(* IEC 61131-3 sources: POC_HINCAPIE/Project/SIEMENS/DIGSI/Guadalupe/TMP/CFC/7344242.18124 (part 2) *)

     AND10_9             (X1 := OR10_7.Y,
                          X2 := AND10_6.Y,
                          X3 := 1,
                          X4 := 1,
                          X5 := 1,
                          X6 := 1,
                          X7 := 1,
                          X8 := 1,
                          X9 := 1,
                          X10 := 1);

     AND10_10            (X1 := AND10_2.Y,
                          X2 := AND10_6.Y,
                          X3 := 1,
                          X4 := 1,
                          X5 := 1,
                          X6 := 1,
                          X7 := 1,
                          X8 := 1,
                          X9 := 1,
                          X10 := 1);

     AND10_11            (X1 := AND10_6.Y,
                          X2 := AND10_3.Y,
                          X3 := 1,
                          X4 := 1,
                          X5 := 1,
                          X6 := 1,
                          X7 := 1,
                          X8 := 1,
                          X9 := 1,
                          X10 := 1);

     OR10_12             (X1 := AND10_9.Y,
                          X2 := AND10_8.Y,
                          X3 := 0,
                          X4 := 0,
                          X5 := 0,
                          X6 := 0,
                          X7 := 0,
                          X8 := 0,
                          X9 := 0,
                          X10 := 0);

     AND10_13            (X1 := EXV_SPS_0144.VAL(* POSITION := 39*79: SIZE := 32* -1:   *) ,
                          X2 := EXV_SPS_0148.VAL(* POSITION := 40*80: SIZE := 31* -1:   *) ,
                          X3 := OR10_1.Y,
                          X4 := 1,
                          X5 := 1,
                          X6 := 1,
                          X7 := 1,
                          X8 := 1,
                          X9 := 1,
                          X10 := 1);

     EXV_SPS_0123        (LNK := 123,
                          VAL := AND10_3.Y(* POSITION := 53*59: SIZE := 32* -1:   *) );
     EXV_SPS_0124        (LNK := 124,
                          VAL := AND10_11.Y(* POSITION := 119*19: SIZE := 34* -1:   *) );
     EXV_SPS_0125        (LNK := 125,
                          VAL := AND10_2.Y(* POSITION := 65*7: SIZE := 32* -1:   *) );
     EXV_SPS_0126        (LNK := 126,
                          VAL := AND10_10.Y(* POSITION := 119*12: SIZE := 34* -1:   *) );
     EXV_SPS_0127        (LNK := 127,
                          VAL := OR10_7.Y(* POSITION := 117*26: SIZE := 31* -1:   *) );
     EXV_SPS_0128        (LNK := 128,
                          VAL := AND10_9.Y(* POSITION := 117*37: SIZE := 34* -1:   *) );
     EXV_SPS_0129        (LNK := 129,
                          VAL := OR10_12.Y(* POSITION := 112*56: SIZE := 34* -1:   *) );
     EXV_SPS_0130        (LNK := 130,
                          VAL := AND10_8.Y(* POSITION := 93*67: SIZE := 32* -1:   *) );
     EXV_SPS_0131        (LNK := 131,
                          VAL := AND10_13.Y(* POSITION := 96*79: SIZE := 29* -1:   *) );
     EXV_SPS_0142        (LNK := 142,
                          VAL := AND10_8.Y(* POSITION := 93*66: SIZE := 34* -1:   *) );
     EXV_SPS_0143        (LNK := 143,
                          VAL := AND10_9.Y(* POSITION := 117*36: SIZE := 35* -1:   *) );
     EXV_SPS_0147        (LNK := 147,
                          VAL := OR10_1.Y(* POSITION := 97*87: SIZE := 31* -1:   *) );
     EXV_SPS_0149        (LNK := 149,
                          VAL := OR10_12.Y(* POSITION := 110*55: SIZE := 38* -1:   *) );
     EXV_SPS_0151        (LNK := 151,
                          VAL := AND10_5.Y(* POSITION := -1*-1: SIZE := 33* -1:   *) );

(* COMMENT_TEXT;{X=70,Y=2};{Width=33, Height=2};FontSize := 12,LineColor := 0,LineWidth := 0,Alignment := Near,AutoWrap := True,BackColor := -16711681,Background := False,TextColor := 0,WallpaperGamma := 100,PartitionID := 1,;Enclavamiento Cierre Interruptor de 13.8 kV *)
(* COMMENT_TEXT;{X=12,Y=6};{Width=21, Height=2};FontSize := 12,LineColor := 0,LineWidth := 0,Alignment := Near,AutoWrap := True,BackColor := -16711681,Background := False,TextColor := 0,WallpaperGamma := 100,PartitionID := 1,;Interruptor Mantenimiento *)
(* COMMENT_TEXT;{X=18,Y=46};{Width=17, Height=2};FontSize := 12,LineColor := 0,LineWidth := 0,Alignment := Near,AutoWrap := True,BackColor := -16711681,Background := False,TextColor := 0,WallpaperGamma := 100,PartitionID := 1,;Interruptor Operación *)
(* COMMENT_TEXT;{X=33,Y=61};{Width=37, Height=2};FontSize := 12,LineColor := 0,LineWidth := 0,Alignment := Near,AutoWrap := True,BackColor := -16711681,Background := False,TextColor := 0,WallpaperGamma := 100,PartitionID := 1,;Enclavamientos Apertura Interruptor de 13.8 kV *)

END_PROGRAM

                                                  (* ---------- Program : CHART_dc33a26f_dd72_4905_a63e_bf494be4a4b3 ----------  *)

PROGRAM CHART_dc33a26f_dd72_4905_a63e_bf494be4a4b3
{COMMENT := "Enclavamiento Q1 - Q2";DESC := "";}
(* ChartLayout;PageSize := A4,Rows := 3,Columns := 2,MarginMode := WithoutMargins,MarginSize := 37,MarginLines := 1 *)
(* PartitionInfo;Id := 1,Name := Partition_1,Comment :=   *)
VAR

     (* IO_IOVISIBILITY;OR10_1;X3:X4:X5:X6:X7:X8:X9:X10: *)

     (* PartitionInfo;PartitionID OR10_1;1  *)
OR10_1          { COMMENT := 'or10_4'; POSITION := 49,39; SIZE := 12, 12; } :OR10;

     (* IO_IOVISIBILITY;OR10_2;X3:X4:X5:X6:X7:X8:X9:X10: *)

     (* PartitionInfo;PartitionID OR10_2;1  *)
OR10_2          { COMMENT := 'or10_9'; POSITION := 49,113; SIZE := 12, 12; } :OR10;

     (* IO_IOVISIBILITY;AND10_3;X3:X4:X5:X6:X7:X8:X9:X10: *)

     (* PartitionInfo;PartitionID AND10_3;1  *)
AND10_3         { COMMENT := 'and10_1'; POSITION := 48,6; SIZE := 12, 12; } :AND10;

     (* IO_IOVISIBILITY;AND10_4;X4:X5:X6:X7:X8:X9:X10: *)

     (* PartitionInfo;PartitionID AND10_4;1  *)
AND10_4         { COMMENT := 'and10_2'; POSITION := 48,14; SIZE := 12, 12; } :AND10;

     (* IO_IOVISIBILITY;AND10_5;X3:X4:X5:X6:X7:X8:X9:X10: *)

     (* PartitionInfo;PartitionID AND10_5;1  *)
AND10_5         { COMMENT := 'and10_5'; POSITION := 49,81; SIZE := 12, 12; } :AND10;

     (* IO_IOVISIBILITY;AND10_6;X4:X5:X6:X7:X8:X9:X10: *)

     (* PartitionInfo;PartitionID AND10_6;1  *)
AND10_6         { COMMENT := 'and10_6'; POSITION := 49,89; SIZE := 12, 12; } :AND10;

     (* IO_IOVISIBILITY;AND10_7;X6:X7:X8:X9:X10: *)

     (* PartitionInfo;PartitionID AND10_7;1  *)
AND10_7         { COMMENT := 'and10_4'; POSITION := 49,29; SIZE := 12, 12; } :AND10;

     (* IO_IOVISIBILITY;AND10_8;X6:X7:X8:X9:X10: *)

     (* PartitionInfo;PartitionID AND10_8;1  *)
AND10_8         { COMMENT := 'and10_22'; POSITION := 49,103; SIZE := 12, 12; } :AND10;

     (* IO_IOVISIBILITY;OR10_9;X3:X4:X5:X6:X7:X8:X9:X10: *)

     (* PartitionInfo;PartitionID OR10_9;1  *)
OR10_9          { COMMENT := 'or10_1'; POSITION := 70,22; SIZE := 12, 12; } :OR10;

     (* IO_IOVISIBILITY;OR10_10;X3:X4:X5:X6:X7:X8:X9:X10: *)

     (* PartitionInfo;PartitionID OR10_10;1  *)
OR10_10         { COMMENT := 'or10_2'; POSITION := 69,95; SIZE := 12, 12; } :OR10;

     (* IO_IOVISIBILITY;AND10_11;X3:X4:X5:X6:X7:X8:X9:X10: *)

     (* PartitionInfo;PartitionID AND10_11;1  *)
AND10_11        { COMMENT := 'and10_3'; POSITION := 89,28; SIZE := 12, 12; } :AND10;

     (* IO_IOVISIBILITY;AND10_12;X3:X4:X5:X6:X7:X8:X9:X10: *)

     (* PartitionInfo;PartitionID AND10_12;1  *)
AND10_12        { COMMENT := 'and10_7'; POSITION := 93,102; SIZE := 12, 12; } :AND10;

     (* 0152 - GDL69TRF2BCU_.Application.FG1_UserDef.FB2_Universal.PerQ1 *)
     EXV_SPS_0152   {COMMENT := "GDL69TRF2BCU_.Application.FG1_UserDef.FB2_Universal.PerQ1";DESC := "0##Application#Usuario#Logicas#Permisivo Q1##1";}:OEXV_BO_SPS;

     (* 0153 - GDL69TRF2BCU_.Application.FG1_Switch.FB1_XSWI.Pos.DPC_StatusOff *)
     EXV_SPS_0153   {COMMENT := "GDL69TRF2BCU_.Application.FG1_Switch.FB1_XSWI.Pos.DPC_StatusOff";DESC := "0##Application#6T4-Q1#Disconnector#Position#open##1";}:IEXV_SPS_BO;

     (* 0154 - GDL69TRF2BCU_.Application.FG1_Breaker_3pol.FB1_XCBR.Pos.DPC_StatusOff *)
     EXV_SPS_0154   {COMMENT := "GDL69TRF2BCU_.Application.FG1_Breaker_3pol.FB1_XCBR.Pos.DPC_StatusOff";DESC := "0##Application#6T4-Q0#Circuit break.#Position#open##1";}:IEXV_SPS_BO;

     (* 0155 - GDL69TRF2BCU_.Application.FG1_Switch.FB1_XSWI.Pos.DPC_StatusOn *)
     EXV_SPS_0155   {COMMENT := "GDL69TRF2BCU_.Application.FG1_Switch.FB1_XSWI.Pos.DPC_StatusOn";DESC := "0##Application#6T4-Q1#Disconnector#Position#closed##1";}:IEXV_SPS_BO;

     (* 0156 - GDL69TRF2BCU_.Application.FG2_Switch.FB1_XSWI.Pos.DPC_StatusOn *)
     EXV_SPS_0156   {COMMENT := "GDL69TRF2BCU_.Application.FG2_Switch.FB1_XSWI.Pos.DPC_StatusOn";DESC := "0##Application#6T4-Q2#Disconnector#Position#closed##1";}:IEXV_SPS_BO;

     (* 0157 - GDL69TRF2BCU_.Application.FG2_Switch.FB1_XSWI.Pos.DPC_StatusOff *)
     EXV_SPS_0157   {COMMENT := "GDL69TRF2BCU_.Application.FG2_Switch.FB1_XSWI.Pos.DPC_StatusOff";DESC := "0##Application#6T4-Q2#Disconnector#Position#open##1";}:IEXV_SPS_BO;

     (* 0158 - GDL69TRF2BCU_.Application.FG1_Switch.FB1_CILO.EnaOpnFix *)
     EXV_SPS_0158   {COMMENT := "GDL69TRF2BCU_.Application.FG1_Switch.FB1_CILO.EnaOpnFix";DESC := "0##Application#6T4-Q1#Interlocking#>Enable opening(fixed)##1";}:OEXV_BO_SPS;

     (* 0159 - GDL69TRF2BCU_.Application.FG1_Switch.FB1_CILO.EnaClsFix *)
     EXV_SPS_0159   {COMMENT := "GDL69TRF2BCU_.Application.FG1_Switch.FB1_CILO.EnaClsFix";DESC := "0##Application#6T4-Q1#Interlocking#>Enable closing (fixed)##1";}:OEXV_BO_SPS;

     (* 0160 - GDL69TRF2BCU_.Application.FG1_UserDef.FB1_Universal.SPS43 *)
     EXV_SPS_0160   {COMMENT := "GDL69TRF2BCU_.Application.FG1_UserDef.FB1_Universal.SPS43";DESC := "0##Application#Usuario#Entradas#Selector Remoto Q1##1";}:IEXV_SPS_BO;

     (* 0161 - GDL69TRF2BCU_.Application.FG1_UserDef.FB1_Universal.FaVcdQ1 *)
     EXV_SPS_0161   {COMMENT := "GDL69TRF2BCU_.Application.FG1_UserDef.FB1_Universal.FaVcdQ1";DESC := "0##Application#Usuario#Entradas#FVCD Q1##1";}:IEXV_SPS_BO;

     (* 0162 - GDL69TRF2BCU_.Application.FG1_UserDef.FB1_Universal.FaVcdSecc *)
     EXV_SPS_0162   {COMMENT := "GDL69TRF2BCU_.Application.FG1_UserDef.FB1_Universal.FaVcdSecc";DESC := "0##Application#Usuario#Entradas#FVCD Cto Control Seccionadores##1";}:IEXV_SPS_BO;

     (* 0163 - GDL69TRF2BCU_.Application.FG2_Switch.FB1_CILO.EnaOpnFix *)
     EXV_SPS_0163   {COMMENT := "GDL69TRF2BCU_.Application.FG2_Switch.FB1_CILO.EnaOpnFix";DESC := "0##Application#6T4-Q2#Interlocking#>Enable opening(fixed)##1";}:OEXV_BO_SPS;

     (* 0164 - GDL69TRF2BCU_.Application.FG2_Switch.FB1_CILO.EnaClsFix *)
     EXV_SPS_0164   {COMMENT := "GDL69TRF2BCU_.Application.FG2_Switch.FB1_CILO.EnaClsFix";DESC := "0##Application#6T4-Q2#Interlocking#>Enable closing (fixed)##1";}:OEXV_BO_SPS;

     (* 0165 - GDL69TRF2BCU_.Application.FG1_UserDef.FB1_Universal.FaVcdQ2 *)
     EXV_SPS_0165   {COMMENT := "GDL69TRF2BCU_.Application.FG1_UserDef.FB1_Universal.FaVcdQ2";DESC := "0##Application#Usuario#Entradas#FVCD Q2##1";}:IEXV_SPS_BO;

     (* 0166 - GDL69TRF2BCU_.Application.FG1_UserDef.FB1_Universal.SPS49 *)
     EXV_SPS_0166   {COMMENT := "GDL69TRF2BCU_.Application.FG1_UserDef.FB1_Universal.SPS49";DESC := "0##Application#Usuario#Entradas#Selector Remoto Q2##1";}:IEXV_SPS_BO;

     (* 0167 - GDL69TRF2BCU_.Application.FG1_Breaker_3pol.FB1_XCBR.Pos.DPC_StatusOn *)
     EXV_SPS_0167   {COMMENT := "GDL69TRF2BCU_.Application.FG1_Breaker_3pol.FB1_XCBR.Pos.DPC_StatusOn";DESC := "0##Application#6T4-Q0#Circuit break.#Position#closed##1";}:IEXV_SPS_BO;

     (* 0168 - GDL69TRF2BCU_.Application.FG1_UserDef.FB1_Universal.SPS113 *)
     EXV_SPS_0168   {COMMENT := "GDL69TRF2BCU_.Application.FG1_UserDef.FB1_Universal.SPS113";DESC := "0##Application#Usuario#Entradas#Bahia Acople Cerrada##1";}:IEXV_SPS_BO;

     (* 0169 - GDL69TRF2BCU_.Application.FG1_UserDef.FB2_Universal.PerQ1AcpCrdo *)
     EXV_SPS_0169   {COMMENT := "GDL69TRF2BCU_.Application.FG1_UserDef.FB2_Universal.PerQ1AcpCrdo";DESC := "0##Application#Usuario#Logicas#Permisivo Q1 Acople Cerrado##1";}:OEXV_BO_SPS;

     (* 0170 - GDL69TRF2BCU_.Application.FG1_UserDef.FB2_Universal.OrQ1 *)
     EXV_SPS_0170   {COMMENT := "GDL69TRF2BCU_.Application.FG1_UserDef.FB2_Universal.OrQ1";DESC := "0##Application#Usuario#Logicas#Or Q1##1";}:OEXV_BO_SPS;

     (* 0171 - GDL69TRF2BCU_.Application.FG1_UserDef.FB2_Universal.PerQ1Gral *)
     EXV_SPS_0171   {COMMENT := "GDL69TRF2BCU_.Application.FG1_UserDef.FB2_Universal.PerQ1Gral";DESC := "0##Application#Usuario#Logicas#Permisivo General Q1##1";}:OEXV_BO_SPS;

     (* 0172 - GDL69TRF2BCU_.Application.FG1_UserDef.FB2_Universal.OrQ2 *)
     EXV_SPS_0172   {COMMENT := "GDL69TRF2BCU_.Application.FG1_UserDef.FB2_Universal.OrQ2";DESC := "0##Application#Usuario#Logicas#Or Q2##1";}:OEXV_BO_SPS;

     (* 0173 - GDL69TRF2BCU_.Application.FG1_UserDef.FB2_Universal.PerQ2AcpCrdo *)
     EXV_SPS_0173   {COMMENT := "GDL69TRF2BCU_.Application.FG1_UserDef.FB2_Universal.PerQ2AcpCrdo";DESC := "0##Application#Usuario#Logicas#Permisivo Q2 Acople Cerrado##1";}:OEXV_BO_SPS;

     (* 0174 - GDL69TRF2BCU_.Application.FG1_UserDef.FB2_Universal.PerQ2Gral *)
     EXV_SPS_0174   {COMMENT := "GDL69TRF2BCU_.Application.FG1_UserDef.FB2_Universal.PerQ2Gral";DESC := "0##Application#Usuario#Logicas#Permisivo General Q2##1";}:OEXV_BO_SPS;

     (* 0175 - GDL69TRF2BCU_.Application.FG1_UserDef.FB2_Universal.PerQ2 *)
     EXV_SPS_0175   {COMMENT := "GDL69TRF2BCU_.Application.FG1_UserDef.FB2_Universal.PerQ2";DESC := "0##Application#Usuario#Logicas#Permisivo Q2##1";}:OEXV_BO_SPS;

     (* 0176 - GDL69TRF2BCU_.Application.FG1_UserDef.FB1_Universal.ManiInsertQ1 *)
     EXV_SPS_0176   {COMMENT := "GDL69TRF2BCU_.Application.FG1_UserDef.FB1_Universal.ManiInsertQ1";DESC := "0##Application#Usuario#Entradas#Manivela Insertada Q1##1";}:IEXV_SPS_BO;

     (* 0177 - GDL69TRF2BCU_.Application.FG1_UserDef.FB1_Universal.ManiInsertQ2 *)
     EXV_SPS_0177   {COMMENT := "GDL69TRF2BCU_.Application.FG1_UserDef.FB1_Universal.ManiInsertQ2";DESC := "0##Application#Usuario#Entradas#Manivela Insertada Q2##1";}:IEXV_SPS_BO;
END_VAR

     EXV_SPS_0153        (LNK := 153);

     EXV_SPS_0154        (LNK := 154);

     EXV_SPS_0155        (LNK := 155);

     EXV_SPS_0156        (LNK := 156);

     EXV_SPS_0157        (LNK := 157);

     EXV_SPS_0160        (LNK := 160);

     EXV_SPS_0161        (LNK := 161);

     EXV_SPS_0162        (LNK := 162);

     EXV_SPS_0165        (LNK := 165);

     EXV_SPS_0166        (LNK := 166);

     EXV_SPS_0167        (LNK := 167);

     EXV_SPS_0168        (LNK := 168);

     EXV_SPS_0176        (LNK := 176);

     EXV_SPS_0177        (LNK := 177);

     OR10_1              (X1 := EXV_SPS_0153.VAL(* POSITION := 13*42: SIZE := 30* -1:   *) ,
                          X2 := EXV_SPS_0155.VAL(* POSITION := 12*43: SIZE := 31* -1:   *) ,
                          X3 := 0,
                          X4 := 0,
                          X5 := 0,
                          X6 := 0,
                          X7 := 0,
                          X8 := 0,
                          X9 := 0,
                          X10 := 0);

     OR10_2              (X1 := EXV_SPS_0157.VAL(* POSITION := 13*116: SIZE := 30* -1:   *) ,
                          X2 := EXV_SPS_0156.VAL(* POSITION := 12*117: SIZE := 31* -1:   *) ,
                          X3 := 0,
                          X4 := 0,
                          X5 := 0,
                          X6 := 0,
                          X7 := 0,
                          X8 := 0,
                          X9 := 0,
                          X10 := 0);

     AND10_3             (X1 := EXV_SPS_0157.VAL(* POSITION := 12*9: SIZE := 30* -1:   *) ,
                          X2 := EXV_SPS_0154.VAL(* POSITION := 11*10: SIZE := 31* -1:   *) ,
                          X3 := 1,
                          X4 := 1,
                          X5 := 1,
                          X6 := 1,
                          X7 := 1,
                          X8 := 1,
                          X9 := 1,
                          X10 := 1);

     AND10_4             (X1 := EXV_SPS_0156.VAL(* POSITION := 11*17: SIZE := 31* -1:   *) ,
                          X2 := EXV_SPS_0167.VAL(* POSITION := 10*18: SIZE := 32* -1:   *) ,
                          X3 := EXV_SPS_0168.VAL(* POSITION := 10*19: SIZE := 32* -1:   *) ,
                          X4 := 1,
                          X5 := 1,
                          X6 := 1,
                          X7 := 1,
                          X8 := 1,
                          X9 := 1,
                          X10 := 1);

     AND10_5             (X1 := EXV_SPS_0153.VAL(* POSITION := 13*84: SIZE := 30* -1:   *) ,
                          X2 := EXV_SPS_0154.VAL(* POSITION := 12*85: SIZE := 31* -1:   *) ,
                          X3 := 1,
                          X4 := 1,
                          X5 := 1,
                          X6 := 1,
                          X7 := 1,
                          X8 := 1,
                          X9 := 1,
                          X10 := 1);

     AND10_6             (X1 := EXV_SPS_0155.VAL(* POSITION := 10*92: SIZE := 31* -1:   *) ,
                          X2 := EXV_SPS_0167.VAL(* POSITION := 9*93: SIZE := 32* -1:   *) ,
                          X3 := EXV_SPS_0168.VAL(* POSITION := 9*94: SIZE := 32* -1:   *) ,
                          X4 := 1,
                          X5 := 1,
                          X6 := 1,
                          X7 := 1,
                          X8 := 1,
                          X9 := 1,
                          X10 := 1);

     AND10_7             (X1 := EXV_SPS_0160.VAL(* POSITION := 10*32: SIZE := 31* -1:   *) ,
                          X2 := NOT EXV_SPS_0161.VAL(* POSITION := 16*33: SIZE := 25* -1:   *) ,
                          X3 := NOT EXV_SPS_0162.VAL(* POSITION := 4*34: SIZE := 37* -1:   *) ,
                          X4 := NOT EXV_SPS_0176.VAL(* POSITION := 9*35: SIZE := 32* -1:   *) ,
                          X5 := OR10_1.Y,
                          X6 := 1,
                          X7 := 1,
                          X8 := 1,
                          X9 := 1,
                          X10 := 1);

     AND10_8             (X1 := EXV_SPS_0166.VAL(* POSITION := -1*-1: SIZE := 31* -1:   *) ,
                          X2 := NOT EXV_SPS_0165.VAL(* POSITION := -1*-1: SIZE := 25* -1:   *) ,
                          X3 := NOT EXV_SPS_0162.VAL(* POSITION := -1*-1: SIZE := 37* -1:   *) ,
                          X4 := NOT EXV_SPS_0177.VAL(* POSITION := -1*-1: SIZE := 32* -1:   *) ,
                          X5 := OR10_2.Y,
                          X6 := 1,
                          X7 := 1,
                          X8 := 1,
                          X9 := 1,
                          X10 := 1);

     OR10_9              (X1 := AND10_3.Y,
                          X2 := AND10_4.Y,
                          X3 := 0,
                          X4 := 0,
                          X5 := 0,
                          X6 := 0,
                          X7 := 0,
                          X8 := 0,
                          X9 := 0,
                          X10 := 0);

     OR10_10             (X1 := AND10_5.Y,
                          X2 := AND10_6.Y,
                          X3 := 0,
                          X4 := 0,
                          X5 := 0,
                          X6 := 0,
                          X7 := 0,
                          X8 := 0,
                          X9 := 0,
                          X10 := 0);

     AND10_11            (X1 := OR10_9.Y,
                          X2 := AND10_7.Y,
                          X3 := 1,
                          X4 := 1,
                          X5 := 1,
                          X6 := 1,
                          X7 := 1,
                          X8 := 1,
                          X9 := 1,
                          X10 := 1);

     AND10_12            (X1 := OR10_10.Y,
                          X2 := AND10_8.Y,
                          X3 := 1,
                          X4 := 1,
                          X5 := 1,
                          X6 := 1,
                          X7 := 1,
                          X8 := 1,
                          X9 := 1,
                          X10 := 1);

     EXV_SPS_0152        (LNK := 152,
                          VAL := AND10_3.Y(* POSITION := 67*9: SIZE := 27* -1:   *) );
     EXV_SPS_0158        (LNK := 158,
                          VAL := AND10_11.Y(* POSITION := 108*33: SIZE := 34* -1:   *) );
     EXV_SPS_0159        (LNK := 159,
                          VAL := AND10_11.Y(* POSITION := 108*32: SIZE := 35* -1:   *) );
     EXV_SPS_0163        (LNK := 163,
                          VAL := AND10_12.Y(* POSITION := 112*106: SIZE := 34* -1:   *) );
     EXV_SPS_0164        (LNK := 164,
                          VAL := AND10_12.Y(* POSITION := 112*105: SIZE := 35* -1:   *) );
     EXV_SPS_0169        (LNK := 169,
                          VAL := AND10_4.Y(* POSITION := 68*17: SIZE := 35* -1:   *) );
     EXV_SPS_0170        (LNK := 170,
                          VAL := OR10_9.Y(* POSITION := 89*25: SIZE := 24* -1:   *) );
     EXV_SPS_0171        (LNK := 171,
                          VAL := AND10_11.Y(* POSITION := 108*31: SIZE := 31* -1:   *) );
     EXV_SPS_0172        (LNK := 172,
                          VAL := OR10_10.Y(* POSITION := 88*98: SIZE := 24* -1:   *) );
     EXV_SPS_0173        (LNK := 173,
                          VAL := AND10_6.Y(* POSITION := 68*92: SIZE := 35* -1:   *) );
     EXV_SPS_0174        (LNK := 174,
                          VAL := AND10_12.Y(* POSITION := 112*107: SIZE := 31* -1:   *) );
     EXV_SPS_0175        (LNK := 175,
                          VAL := AND10_5.Y(* POSITION := 68*84: SIZE := 27* -1:   *) );

(* COMMENT_TEXT;{X=43,Y=1};{Width=23, Height=2};FontSize := 12,LineColor := 0,LineWidth := 0,Alignment := Near,AutoWrap := True,BackColor := -16711681,Background := False,TextColor := 0,WallpaperGamma := 100,PartitionID := 1,;Enclavamiento Seccionador Q1 *)
(* COMMENT_TEXT;{X=45,Y=73};{Width=23, Height=2};FontSize := 12,LineColor := 0,LineWidth := 0,Alignment := Near,AutoWrap := True,BackColor := -16711681,Background := False,TextColor := 0,WallpaperGamma := 100,PartitionID := 1,;Enclavamiento Seccionador Q2 *)

END_PROGRAM

                                                  (* ---------- Program : CHART_Enclavamiento_Q9 ----------  *)

PROGRAM CHART_Enclavamiento_Q9
{COMMENT := "Enclavamiento Q9";DESC := "";}
(* ChartLayout;PageSize := A4,Rows := 3,Columns := 2,MarginMode := WithoutMargins,MarginSize := 37,MarginLines := 1 *)
(* PartitionInfo;Id := 1,Name := Partition_1,Comment :=   *)
VAR

     (* IO_IOVISIBILITY;OR10_1;X3:X4:X5:X6:X7:X8:X9:X10: *)

     (* PartitionInfo;PartitionID OR10_1;1  *)
OR10_1          { COMMENT := 'or10_5'; POSITION := 69,22; SIZE := 12, 12; } :OR10;

     (* IO_IOVISIBILITY;AND10_2;X7:X8:X9:X10: *)

     (* PartitionInfo;PartitionID AND10_2;1  *)
AND10_2         { COMMENT := 'and10_8'; POSITION := 69,11; SIZE := 12, 12; } :AND10;

     (* 0178 - GDL69TRF2BCU_.Application.FG1_UserDef.FB2_Universal.PerQ9 *)
     EXV_SPS_0178   {COMMENT := "GDL69TRF2BCU_.Application.FG1_UserDef.FB2_Universal.PerQ9";DESC := "0##Application#Usuario#Logicas#Permisivo Q9##1";}:OEXV_BO_SPS;

     (* 0179 - GDL69TRF2BCU_.Application.FG3_Switch.FB1_XSWI.Pos.DPC_StatusOff *)
     EXV_SPS_0179   {COMMENT := "GDL69TRF2BCU_.Application.FG3_Switch.FB1_XSWI.Pos.DPC_StatusOff";DESC := "0##Application#6T4-Q9#Disconnector#Position#open##1";}:IEXV_SPS_BO;

     (* 0180 - GDL69TRF2BCU_.Application.FG1_Breaker_3pol.FB1_XCBR.Pos.DPC_StatusOff *)
     EXV_SPS_0180   {COMMENT := "GDL69TRF2BCU_.Application.FG1_Breaker_3pol.FB1_XCBR.Pos.DPC_StatusOff";DESC := "0##Application#6T4-Q0#Circuit break.#Position#open##1";}:IEXV_SPS_BO;

     (* 0181 - GDL69TRF2BCU_.Application.FG3_Switch.FB1_XSWI.Pos.DPC_StatusOn *)
     EXV_SPS_0181   {COMMENT := "GDL69TRF2BCU_.Application.FG3_Switch.FB1_XSWI.Pos.DPC_StatusOn";DESC := "0##Application#6T4-Q9#Disconnector#Position#closed##1";}:IEXV_SPS_BO;

     (* 0182 - GDL69TRF2BCU_.Application.FG1_UserDef.FB1_Universal.FaVcdSecc *)
     EXV_SPS_0182   {COMMENT := "GDL69TRF2BCU_.Application.FG1_UserDef.FB1_Universal.FaVcdSecc";DESC := "0##Application#Usuario#Entradas#FVCD Cto Control Seccionadores##1";}:IEXV_SPS_BO;

     (* 0183 - GDL69TRF2BCU_.Application.FG1_UserDef.FB1_Universal.SPS55 *)
     EXV_SPS_0183   {COMMENT := "GDL69TRF2BCU_.Application.FG1_UserDef.FB1_Universal.SPS55";DESC := "0##Application#Usuario#Entradas#Selector Remoto Q9##1";}:IEXV_SPS_BO;

     (* 0184 - GDL69TRF2BCU_.Application.FG1_UserDef.FB1_Universal.FaVcdQ9 *)
     EXV_SPS_0184   {COMMENT := "GDL69TRF2BCU_.Application.FG1_UserDef.FB1_Universal.FaVcdQ9";DESC := "0##Application#Usuario#Entradas#FVCD Q9##1";}:IEXV_SPS_BO;

     (* 0185 - GDL69TRF2BCU_.Application.FG3_Switch.FB1_CILO.EnaClsFix *)
     EXV_SPS_0185   {COMMENT := "GDL69TRF2BCU_.Application.FG3_Switch.FB1_CILO.EnaClsFix";DESC := "0##Application#6T4-Q9#Interlocking#>Enable closing (fixed)##1";}:OEXV_BO_SPS;

     (* 0186 - GDL69TRF2BCU_.Application.FG3_Switch.FB1_CILO.EnaOpnFix *)
     EXV_SPS_0186   {COMMENT := "GDL69TRF2BCU_.Application.FG3_Switch.FB1_CILO.EnaOpnFix";DESC := "0##Application#6T4-Q9#Interlocking#>Enable opening(fixed)##1";}:OEXV_BO_SPS;

     (* 0187 - GDL69TRF2BCU_.Application.FG1_UserDef.FB1_Universal.ManiInsertQ9 *)
     EXV_SPS_0187   {COMMENT := "GDL69TRF2BCU_.Application.FG1_UserDef.FB1_Universal.ManiInsertQ9";DESC := "0##Application#Usuario#Entradas#Manivela Insertada Q9##1";}:IEXV_SPS_BO;
END_VAR

     EXV_SPS_0179        (LNK := 179);

     EXV_SPS_0180        (LNK := 180);

     EXV_SPS_0181        (LNK := 181);

     EXV_SPS_0182        (LNK := 182);

     EXV_SPS_0183        (LNK := 183);

     EXV_SPS_0184        (LNK := 184);

     EXV_SPS_0187        (LNK := 187);

     OR10_1              (X1 := EXV_SPS_0179.VAL(* POSITION := 33*25: SIZE := 30* -1:   *) ,
                          X2 := EXV_SPS_0181.VAL(* POSITION := 32*26: SIZE := 31* -1:   *) ,
                          X3 := 0,
                          X4 := 0,
                          X5 := 0,
                          X6 := 0,
                          X7 := 0,
                          X8 := 0,
                          X9 := 0,
                          X10 := 0);

     AND10_2             (X1 := EXV_SPS_0180.VAL(* POSITION := 32*14: SIZE := 31* -1:   *) ,
                          X2 := EXV_SPS_0183.VAL(* POSITION := 32*15: SIZE := 31* -1:   *) ,
                          X3 := NOT EXV_SPS_0184.VAL(* POSITION := 38*16: SIZE := 25* -1:   *) ,
                          X4 := NOT EXV_SPS_0182.VAL(* POSITION := 26*17: SIZE := 37* -1:   *) ,
                          X5 := NOT EXV_SPS_0187.VAL(* POSITION := -1*-1: SIZE := 32* -1:   *) ,
                          X6 := OR10_1.Y,
                          X7 := 1,
                          X8 := 1,
                          X9 := 1,
                          X10 := 1);

     EXV_SPS_0178        (LNK := 178,
                          VAL := AND10_2.Y(* POSITION := 88*16: SIZE := 27* -1:   *) );
     EXV_SPS_0185        (LNK := 185,
                          VAL := AND10_2.Y(* POSITION := 88*15: SIZE := 35* -1:   *) );
     EXV_SPS_0186        (LNK := 186,
                          VAL := AND10_2.Y(* POSITION := 88*14: SIZE := 34* -1:   *) );

(* COMMENT_TEXT;{X=63,Y=8};{Width=23, Height=2};FontSize := 12,LineColor := 0,LineWidth := 0,Alignment := Near,AutoWrap := True,BackColor := -16711681,Background := False,TextColor := 0,WallpaperGamma := 100,PartitionID := 1,;Enclavamiento Seccionador Q9 *)

END_PROGRAM

CONFIGURATION  PLC_CONTROL
   RESOURCE PLANS { COMMENT := "Txt100_100";} ON CPU32
     TASK EVENT_SLOW     { TICKS := 1300;}(PRIORITY := INTERNAL);
     TASK EVENT_FAST     { TICKS := 255;}(PRIORITY := INTERNAL);
     TASK MEASUREMENT    { TICKS := 2536;}(PRIORITY := INTERNAL);
     TASK INTERLOCKING   { TICKS := 2173;}(PRIORITY := INTERNAL);

     PROGRAM FBI001 WITH EVENT_SLOW:  CHART_Enclavamiento_Q0_69_kV;
     PROGRAM FBI002 WITH EVENT_SLOW:  CHART_Falla_PTs;
     PROGRAM FBI003 WITH EVENT_SLOW:  CHART_Alarmas;
     PROGRAM FBI004 WITH EVENT_SLOW:  CHART_Falla_Goose;
     PROGRAM FBI005 WITH EVENT_SLOW:  CHART_Sincronismo;
     PROGRAM FBI006 WITH EVENT_SLOW:  CHART_2b45b93f_4554_488e_9a6f_110f79ec8d45;
     PROGRAM FBI007 WITH EVENT_SLOW:  CHART_dc33a26f_dd72_4905_a63e_bf494be4a4b3;
     PROGRAM FBI008 WITH EVENT_SLOW:  CHART_Enclavamiento_Q9;

   END_RESOURCE

 END_CONFIGURATION
